# B&R Automation Studio project 02_BASE_PROJECT
Automation Studio 4.9

## Configuration Config1

CPU X20CP1382, AutomationRuntime A4.83, Build 4.1.2, Safety 0.0, Vc V4.73.2

### Task classes (Cpu.sw)
```
Cyclic#1 (cycle 2000 us, tolerance 0 us):
  ComTCP_P <- Libraries.ComTCP.ComTCP_P.prg
  Input_Brid <- Input_Bridge.prg
  Output_Bri <- Output_Bridge.prg
  PLCopen <- PLCopen.prg [disabled]
Cyclic#2:
  LED_IO <- LED_IO.prg
  Master <- Master.prg
  Slave <- Slave.prg
DataObjects: Acp10sys
NcDataObjects: acp10etxen <- acp10etxen.dob, gAxis01a <- gAxis01obj.gAxis01a.dob, gAxis01i <- gAxis01obj.gAxis01i.dob, gAxis02a <- gAxis02obj.gAxis02a.dob, gAxis02i <- gAxis02obj.gAxis02i.dob, MyCam <- MyCam.dob, MyCamBis <- MyCamBis.dob
Binaries: udbdef, FWRules, TCData, arsvcreg, mvLoader, TCLang, acp10cfg, Acp10map, sysconf, Role, User, iomap, ashwd, asfw, arconfig, ashwac, Config, TC
Libraries: Acp10man, Acp10par, NcGlobal, Acp10_MC, sys_lib, brsystem, runtime, Acp10sim, MpAxis, MpBase, MpCom, AsTCP, standard, AsArLog, AsBrStr, ComTCP_L, operator, astime, AsIecCon, My_Library, AsIODiag, fileio, powerlnk, dataobj, arssl
```

### Hardware
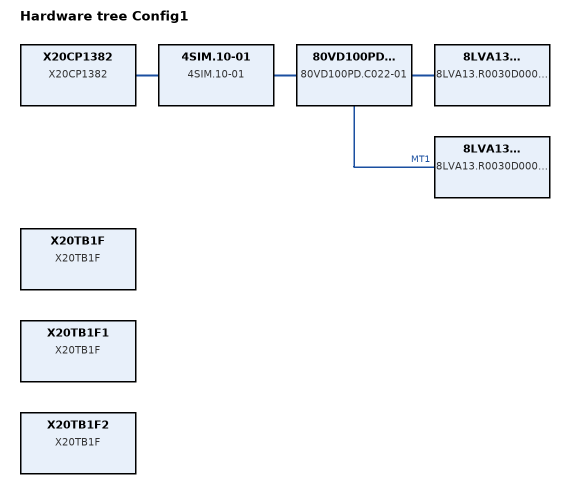
```
4SIM.10-01 : 4SIM.10-01 v1.3.0.0  [PLK1 -> X20CP1382.IF3 (NodeNumber=1) [Cable Type=PowerlinkCable, Length=10, Version=1.0.0.3]; PLK2 -> 80VD100PD.C022-01.PLK1 (NodeNumber=1) [Cable Type=PowerlinkCable, Length=10, Version=1.0.0.3]]
  Supervision = off
80VD100PD.C022-01 : 80VD100PD.C022-01 v2.5.0.0  [PLK1 -> 4SIM.10-01.PLK2 (NodeNumber=2) [Cable Type=PowerlinkCable, Length=10, Version=1.0.0.3]; MT2 -> 8LVA13.R0030D000-0.MT]
  MotionTP = Acp10Arnc0
  AxisIsPeriodic_r1 = on
  Period_r1 = 360
  BothEndSwitchesAreNormallyOpen_r1 = on
  QuickStopIsNormallyOpen_r1 = on
  AxisIsPeriodic_r2 = on
  Period_r2 = 360
  BothEndSwitchesAreNormallyOpen_r2 = on
  QuickStopIsNormallyOpen_r2 = on
8LVA13.R0030D000-0 : 8LVA13.R0030D000-0 v2.2.0.4  [MT -> 80VD100PD.C022-01.MT2]
8LVA13.R0030D000-0a : 8LVA13.R0030D000-0 v2.2.0.4  [MT -> 80VD100PD.C022-01.MT1]
X20CP1382 : X20CP1382 v1.14.0.0  [X1 -> X1.SL; X2 -> X2.SL; X3 -> X3.SL]
  Module X1 (Type=X1, Virtual=true, Version=1.14.0.0)
    Connection (Connector=SS1, TargetModule=X20TB1F, TargetConnector=SS)
    Connection (Connector=SL, TargetModule=X20CP1382, TargetConnector=X1)
  Module X2 (Type=X2, Virtual=true, Version=1.14.0.0)
    Connection (Connector=SS1, TargetModule=X20TB1F1, TargetConnector=SS)
    Connection (Connector=SL, TargetModule=X20CP1382, TargetConnector=X2)
  Module X3 (Type=X3, Virtual=true, Version=1.14.0.0)
    Connection (Connector=SS1, TargetModule=X20TB1F2, TargetConnector=SS)
    Connection (Connector=SL, TargetModule=X20CP1382, TargetConnector=X3)
  Connector IF2:
    ActivateDevice = 1
    Mode = Manual
    InternetAddress = 192.168.0.1
    SubnetMask = 255.255.255.0
    ActivateSnmp = 2
  Connector IF3:
    CycleTime = 2000
  ConfigurationID = UniboTest2024_Config1
  Simulation = 1
  TimerDeviceType = EPLX2X
  TimerDevice = X20CP1382.IF3
  TaskClassIdleTime = 6000
  Cyclic1Duration = 2000
  Cyclic1Tolerance = 0
  ActivateOpcUa = 1
  OpcUaInformationModels_PV_Version = 1
X20TB1F : X20TB1F v1.0.0.0
X20TB1F1 : X20TB1F v1.0.0.0
X20TB1F2 : X20TB1F v1.0.0.0
```

### Acp10map.ncm - X20CP1382/Motion/Acp10map.ncm
```
NcMapping (NcSwId=Acp10)
  NcObject gAxis01 (ModuleId=80VD100PD.C022-01, Type=ncAXIS, Channel=1, AcoposSimulation=Off, InitParameter=gAxis01i, AcoposParameter=gAxis01a, AdditionalData=PLCopen_ModPos="360,1" , Disabled=FALSE, ModuleDisabled=FALSE)
  NcObject gAxis02 (ModuleId=80VD100PD.C022-01, Type=ncAXIS, Channel=2, AcoposSimulation=Off, InitParameter=gAxis02i, AcoposParameter=gAxis02a, AdditionalData=PLCopen_ModPos="360,1" , Disabled=FALSE, ModuleDisabled=FALSE)
  NcObject 80VD100PD.C022-01_ncV_AXIS1 (ModuleId=80VD100PD.C022-01, Type=ncV_AXIS, Channel=1, Disabled=TRUE, ModuleDisabled=FALSE)
  NcObject 80VD100PD.C022-01_ncV_AXIS2 (ModuleId=80VD100PD.C022-01, Type=ncV_AXIS, Channel=2, Disabled=TRUE, ModuleDisabled=FALSE)
```

## Logical view

Binary libraries used (declarations not repeated): operator, runtime, astime, AsIecCon, sys_lib, brsystem, MpAxis, AsTCP, standard, AsArLog, AsBrStr, MpBase, MpCom, AsIODiag, Acp10man, Acp10par, NcGlobal, Acp10sim 5.24.1, Acp10_MC

### Global.var
```iecst
(*Name of Axis*)
VAR
	gAxis01 : ACP10AXIS_typ;
	gAxis02 : ACP10AXIS_typ;
END_VAR
(*Hardware Variables*)
VAR
	Conv_Lock : BOOL;
	Cutter_Lock : BOOL;
	Start_Button : BOOL;
	Stop_Button : BOOL;
	Sensor_Button : BOOL;
	Reset_Button : BOOL;
	Speed : INT;
	Position : INT;
	DI1 : FSM_LED;
	DI2 : FSM_LED;
	DI3 : FSM_LED;
	DI4 : FSM_LED;
	DI5 : FSM_LED;
	DI6 : FSM_LED;
	Display : INT;
END_VAR
(*HMI Variables*)
VAR
	Emergancy_Button_HMI : BOOL;
	Start_Button_HMI : BOOL;
	Stop_Button_HMI : BOOL;
	Sensor_Button_HMI : BOOL;
	Reset_Button_HMI : BOOL;
	Conv_Lock_HMI : BOOL;
	Cutter_Lock_HMI : BOOL;
	Conv_Speed_HMI : REAL;
	Cutter_Speed_HMI : REAL;
	Cutting_Pos_HMI : REAL;
	Cutting_Depth_HMI : REAL;
	Blade_Up_Man_HMI : BOOL;
	Blade_Down_Man_HMI : BOOL;
	Conv_Right_Man_HMI : BOOL;
	Conv_Left_Man_HMI : BOOL;
	Slow_Blade_HMI : BOOL;
	Slow_Conv_HMI : BOOL;
	LED_DI1_HMI : BOOL;
	LED_DI2_HMI : BOOL;
	LED_DI3_HMI : BOOL;
	LED_DI4_HMI : BOOL;
	LED_DI5_HMI : BOOL;
	LED_DI6_HMI : BOOL;
	Dis_Conv_Speed_HMI : REAL;
	Dis_Cut_Speed_HMI : REAL;
	Dis_Cut_Pos_HMI : INT;
	Dis_Cut_Depth_HMI : INT;
	Man_Mode_HMI : BOOL;
	Over_Ride_HMI : BOOL;
END_VAR
(*LED_IO Variables*)
VAR
	Power_Axis : BOOL;
	Home_Axis : BOOL;
	Reset_Command : BOOL;
	Error_Command : BOOL;
	Start_Command : BOOL := FALSE;
	Stop_Command : BOOL := FALSE;
END_VAR
(*Master Variables*)
VAR
	Do_Cut : BOOL;
	Done_Cut : BOOL;
	Master : MpAxisBasic;
	M_Active : BOOL;
	M_Error : BOOL;
	M_Actual_Position : LREAL;
	M_Actual_Velocity : LREAL;
	M_Homed : BOOL;
	M_Powered : BOOL;
	M_Stoped : BOOL;
END_VAR
(*Slave Variables*)
VAR
	Slave : MpAxisBasic;
	Coupling : MpAxisCoupling;
	S_Active : BOOL;
	S_Error : BOOL;
	S_Homed : BOOL;
	S_Powered : BOOL;
	C_Error : BOOL;
	S_Actual_Position : LREAL;
	S_Actual_Velocity : LREAL;
	S_Stoped : BOOL;
END_VAR
(*Input Bridige Variables*)
VAR
	Conv_Speed : REAL;
	Start_Trigger : BOOL;
	Stop_Trigger : BOOL;
	Error_Trigger : BOOL;
	Reset_Trigger : BOOL;
	Conv_Lock_HMI_Trigger : BOOL;
	Cutter_Lock_HMI_Trigger : BOOL;
	Sensor_Trigger : BOOL;
	Conv_Lock_Trigger : BOOL;
	Over_Ride_Trigger : BOOL;
	Cutter_Lock_Trigger : BOOL;
	Slow_Blade_Trigger : BOOL;
	Blade_Up_Man_HMI_Trigger : BOOL;
	Blade_Down_Man_HMI_Trigger : BOOL;
	Conv_Left_Man_HMI_Trigger : BOOL;
	Conv_Right_Man_HMI_Trigger : BOOL;
	Slow_Conv_Trigger : BOOL;
END_VAR
(*Manual Motion Variables*)
VAR
	Manual_Mode_Trigger : BOOL;
	Man_Mode_OFF : BOOL := TRUE;
	Blade_Jog_Velocity : REAL;
	Conv_Jog_Velocity : REAL;
END_VAR
```

- Project.language (not shown)

### Data object Logical/acp10etxen (Ett)

- acp10etxen.ett (not shown)

### Data object Logical/gAxis01obj/gAxis01a (Apt)

#### gAxis01a.apt
```
AcoposParameterTable:
  Root Parameters
```

### gAxis01i.ax
```
InitParameter (Version=5.20.1, NcSwId=ACP10)
  ACP10AXIS_typ:
    dig_in:
      level:
        reference = ncACTIV_HI
        pos_hw_end = ncACTIV_HI
        neg_hw_end = ncACTIV_HI
        trigger1 = ncACTIV_HI
        trigger2 = ncACTIV_HI
    encoder_if:
      parameter:
        count_dir = ncSTANDARD
        scaling:
          load:
            units = 360
            rev_motor = 1
    limit:
      parameter:
        v_pos = 10000.0
        v_neg = 10000.0
        a1_pos = 50000.0
        a2_pos = 50000.0
        a1_neg = 50000.0
        a2_neg = 50000.0
        t_jolt = 0.0
        t_in_pos = 0.0
        pos_sw_end = 2000000000
        neg_sw_end = -2000000000
        ds_warning = 500.0
        ds_stop = 1000.0
        a_stop = 1.0E+30
        dv_stop = 0.0
        dv_stop_mode = ncOFF
    controller:
      mode = ncPOSITION
      position:
        kv = 289.0
        tn = 0.0
        t_predict = 0.0004
        t_total = 0.0004
        p_max = 1.0E+30
        i_max = 0.0
      speed:
        kv = 0.9
        tn = 0.0
        t_filter = 0.0
        isq_filter1:
          type = ncOFF
          a0 = 0.0
          a1 = 0.0
          b0 = 0.0
          b1 = 0.0
          b2 = 0.0
          c0_par_id = 0
          c1_par_id = 0
        isq_filter2:
          type = ncOFF
          a0 = 0.0
          a1 = 0.0
          b0 = 0.0
          b1 = 0.0
          b2 = 0.0
          c0_par_id = 0
          c1_par_id = 0
        isq_filter3:
          type = ncOFF
          a0 = 0.0
          a1 = 0.0
          b0 = 0.0
          b1 = 0.0
          b2 = 0.0
          c0_par_id = 0
          c1_par_id = 0
      uf:
        type = ncLINEAR + ncCORRECTION
        auto_config = ncMOTOR_PAR
        u0 = 0.0
        un = 0.0
        fn = 50.0
        k_f_slip = 0.0
      ff:
        mode = ncSTANDARD
        torque_load = 0.0
        torque_pos = 0.0
        torque_neg = 0.0
        kv_torque = 0.0
        inertia = 0.0
        t_filter_a = 0.0
      fb:
        mode = ncSTANDARD
        speed_mix_ratio = 0.0
        speed_kv = 0.0
      model:
        mass1:
          inertia = 0.0
          viscous_friction = 0.0
        mass2:
          inertia = 0.0
          viscous_friction = 0.0
          stiffness = 0.0
          damping = 0.0
    move:
      stop:
        parameter[0]:
          decel_ramp = ncA_LIMIT
          controller = ncON
        parameter[1]:
          decel_ramp = ncA_LIMIT
          controller = ncON
        parameter[2]:
          decel_ramp = ncA_LIMIT
          controller = ncON
        parameter[3]:
          decel_ramp = ncA_LIMIT
          controller = ncON
        quickstop:
          decel_ramp = ncA_LIMIT
          t_jolt = 0.0
        drive_error:
          decel_ramp = ncA_LIMIT
      homing:
        parameter:
          s = 0
          v_switch = 5000.0
          v_trigger = 500.0
          a = 50000.0
          mode = ncDIRECT
          edge_sw = ncPOSITIVE
          start_dir = ncPOSITIVE
          trigg_dir = ncPOSITIVE
          ref_pulse = ncOFF
          fix_dir = ncOFF
          tr_s_block = 0.0
          torque_lim = 0.0
          ds_block = 0.0
          ds_stop = 0.0
      basis:
        parameter:
          v_pos = 5000.0
          v_neg = 5000.0
          a1_pos = 50000.0
          a2_pos = 50000.0
          a1_neg = 50000.0
          a2_neg = 50000.0
    message:
      text:
        parameter:
          format = ncBREAK
          columns = 80
          data_modul = acp10etxen
```

- Data object Logical/gAxis02obj/gAxis02a (Apt) (no source held here)

### gAxis02i.ax
```
InitParameter (Version=5.20.1, NcSwId=Acp10)
  ACP10AXIS_typ:
    dig_in:
      level:
        reference = ncACTIV_HI
        pos_hw_end = ncACTIV_HI
        neg_hw_end = ncACTIV_HI
        trigger1 = ncACTIV_HI
        trigger2 = ncACTIV_HI
    encoder_if:
      parameter:
        count_dir = ncSTANDARD
        scaling:
          load:
            units = 360
            rev_motor = 1
    limit:
      parameter:
        v_pos = 10000
        v_neg = 10000
        a1_pos = 50000
        a2_pos = 50000
        a1_neg = 50000
        a2_neg = 50000
        t_jolt = 0
        t_in_pos = 0
        pos_sw_end = 2000000000
        neg_sw_end = -2000000000
        ds_warning = 500
        ds_stop = 1000
        a_stop = 1.0e30
        dv_stop = 0
        dv_stop_mode = ncOFF
    controller:
      mode = ncPOSITION
      position:
        kv = 289.0
        tn = 0
        t_predict = 0.0004
        t_total = 0.0004
        p_max = 1.0e30
        i_max = 0
      speed:
        kv = 0.9
        tn = 0
        t_filter = 0.0
        isq_filter1:
          type = ncOFF
          a0 = 0.0
          a1 = 0.0
          b0 = 0.0
          b1 = 0.0
          b2 = 0.0
          c0_par_id = 0
          c1_par_id = 0
        isq_filter2:
          type = ncOFF
          a0 = 0.0
          a1 = 0.0
          b0 = 0.0
          b1 = 0.0
          b2 = 0.0
          c0_par_id = 0
          c1_par_id = 0
        isq_filter3:
          type = ncOFF
          a0 = 0.0
          a1 = 0.0
          b0 = 0.0
          b1 = 0.0
          b2 = 0.0
          c0_par_id = 0
          c1_par_id = 0
      uf:
        type = ncLINEAR + ncCORRECTION
        auto_config = ncMOTOR_PAR
        u0 = 0
        un = 0
        fn = 50.0
        k_f_slip = 0
      ff:
        mode = ncSTANDARD
        torque_load = 0.0
        torque_pos = 0.0
        torque_neg = 0.0
        kv_torque = 0.0
        inertia = 0.0
        t_filter_a = 0.0
      fb:
        mode = ncSTANDARD
        speed_mix_ratio = 0.0
        speed_kv = 2.0
      model:
        mass1:
          inertia = 0
          viscous_friction = 0
        mass2:
          inertia = 0
          viscous_friction = 0
          stiffness = 0
          damping = 0
    move:
      stop:
        parameter[0]:
          decel_ramp = ncA_LIMIT
          controller = ncON
        parameter[1]:
          decel_ramp = ncA_LIMIT
          controller = ncON
        parameter[2]:
          decel_ramp = ncA_LIMIT
          controller = ncON
        parameter[3]:
          decel_ramp = ncA_LIMIT
          controller = ncON
        quickstop:
          decel_ramp = ncA_LIMIT
          t_jolt = 0
        drive_error:
          decel_ramp = ncA_LIMIT
      homing:
        parameter:
          s = 0
          v_switch = 5000
          v_trigger = 500
          a = 50000
          mode = ncDIRECT
          edge_sw = ncPOSITIVE
          start_dir = ncPOSITIVE
          trigg_dir = ncPOSITIVE
          ref_pulse = ncOFF
          fix_dir = ncOFF
          tr_s_block = 0
          torque_lim = 0
          ds_block = 0
          ds_stop = 0
      basis:
        parameter:
          v_pos = 5000
          v_neg = 5000
          a1_pos = 50000
          a2_pos = 50000
          a1_neg = 50000
          a2_neg = 50000
    message:
      text:
        parameter:
          format = ncBREAK
          columns = 80
          data_modul = acp10etxen
```

### Program Logical/Input_Bridge

#### Main.st
```iecst
PROGRAM _INIT
	(* Insert code here *)
	//Initial Parameters

	Conv_Speed 		:= 100.0;

END_PROGRAM

PROGRAM _CYCLIC

	IF DiagCpuIsSimulated() THEN
		(* For Simulation *)
		//Operator
		//LED_IO Bridge
		Start_Trigger 			:= ComTCP_SimInputs.Start_Button_ButtonPress 		OR Start_Button_HMI;
		Stop_Trigger 			:= ComTCP_SimInputs.Stop_Button_ButtonPress 		OR Stop_Button_HMI;
		Error_Trigger 			:= ComTCP_SimInputs.Emergency_Button_ButtonToggle 	OR Emergancy_Button_HMI OR M_Error OR S_Error OR C_Error;
		Reset_Trigger 			:= ComTCP_SimInputs.White_Button_ButtonPress 		OR Reset_Button_HMI;
		Sensor_Trigger 			:= ComTCP_SimInputs.Yellow_Button_ButtonPress 		OR Sensor_Button_HMI;
		Conv_Lock_HMI_Trigger 	:= Conv_Lock_HMI;
		Cutter_Lock_HMI_Trigger := Cutter_Lock_HMI;

		IF Conv_Lock_HMI_Trigger THEN
			IF Conv_Speed_HMI < 10 THEN
				Conv_Speed 	:= 10;
			ELSE
				Conv_Speed 	:= Conv_Speed_HMI;
			END_IF
		END_IF

		//Manual Motion
		Manual_Mode_Trigger 		:= Man_Mode_HMI;
		Slow_Blade_Trigger 			:= Slow_Blade_HMI;
		Slow_Conv_Trigger 			:= Slow_Conv_HMI;
		Blade_Up_Man_HMI_Trigger 	:= Blade_Up_Man_HMI;
		Blade_Down_Man_HMI_Trigger 	:= Blade_Down_Man_HMI;
		Conv_Left_Man_HMI_Trigger 	:= Conv_Left_Man_HMI;
		Conv_Right_Man_HMI_Trigger 	:= Conv_Right_Man_HMI;

		IF Slow_Blade_Trigger THEN
			Blade_Jog_Velocity := 5.0;
		ELSE
			Blade_Jog_Velocity := 100.0;
		END_IF

		IF Slow_Conv_Trigger THEN
			Conv_Jog_Velocity := 5.0;
		ELSE
			Conv_Jog_Velocity := 100.0;
		END_IF

	ELSE
		(* For Actual Setup *)
		Start_Trigger 			:= Start_Button 		OR Start_Button_HMI;
		Stop_Trigger 			:= Stop_Button 			OR Stop_Button_HMI;
		Error_Trigger 			:= Emergancy_Button_HMI OR M_Error OR S_Error;
		Reset_Trigger 			:= Reset_Button 		OR Reset_Button_HMI;
		Sensor_Trigger 			:= Sensor_Button 		OR Sensor_Button_HMI;
		Conv_Lock_HMI_Trigger	:= Conv_Lock_HMI;
		Conv_Lock_HMI_Trigger 	:= Conv_Lock;
		Over_Ride_Trigger 		:= Over_Ride_HMI;
		IF Over_Ride_Trigger THEN
			IF Conv_Lock_HMI_Trigger THEN
				IF Conv_Speed_HMI < 10 THEN
					Conv_Speed 	:= 10;
				ELSE
					Conv_Speed 	:= Conv_Speed_HMI;
				END_IF
			END_IF
		ELSE
			IF Conv_Lock_Trigger THEN
				Conv_Speed 		:= (Speed*3000/32767);
			END_IF
		END_IF

		//Manual Motion
		Manual_Mode_Trigger 		:= Man_Mode_HMI;
		Slow_Blade_Trigger 			:= Slow_Blade_HMI;
		Slow_Conv_Trigger 			:= Slow_Conv_HMI;
		Blade_Up_Man_HMI_Trigger 	:= Blade_Up_Man_HMI;
		Blade_Down_Man_HMI_Trigger 	:= Blade_Down_Man_HMI;
		Conv_Left_Man_HMI_Trigger	:= Conv_Left_Man_HMI;
		Conv_Right_Man_HMI_Trigger 	:= Conv_Right_Man_HMI;
		IF Slow_Blade_Trigger THEN
			Blade_Jog_Velocity := 5.0;
		ELSE
			Blade_Jog_Velocity := 100.0;
		END_IF

		IF Slow_Conv_Trigger THEN
			Conv_Jog_Velocity := 5.0;
		ELSE
			Conv_Jog_Velocity := 100.0;
		END_IF

	END_IF

END_PROGRAM

PROGRAM _EXIT
	(* Insert code here *)

END_PROGRAM
```

### Program Logical/LED_IO

#### Main.st
```iecst
PROGRAM _INIT
	(* Insert code here *)

END_PROGRAM

PROGRAM _CYCLIC
	(* Insert code here *)
	CASE State OF
		0: //Initiation
			DI1(LED_State := 'off');
			DI2(LED_State := 'off');
			DI3(LED_State := 'off');
			DI4(LED_State := 'off');
			DI5(LED_State := 'off');
			DI6(LED_State := 'off');

			IF M_Active AND S_Active AND Man_Mode_OFF THEN
				State := 2;
			END_IF

		1: //Error

			DI1(LED_State := 'off');
			DI2(LED_State := 'off');
			DI3(LED_State := 'off');
			DI4(LED_State := 'off');
			DI5(LED_State := 'off');
			DI6(LED_State := 'blink');

			Error_Command 	:= TRUE;
			Start_Command 	:= FALSE;
			Stop_Command 	:= TRUE;
			Power_Axis 		:= FALSE;

			IF Reset_Trigger THEN
				Reset_Command 	:= TRUE;
				IF NOT Error_Trigger THEN
					Reset_Command 	:= FALSE;
					State 			:= 2;
				END_IF
			END_IF

		2: //Disabled

			DI1(LED_State := 'on');
			DI2(LED_State := 'on');
			DI3(LED_State := 'on');
			DI4(LED_State := 'on');
			DI5(LED_State := 'on');
			DI6(LED_State := 'on');

			IF Reset_Trigger THEN
				Power_Axis 	:= TRUE;
			END_IF

			IF Error_Trigger THEN
				State := 1;
			END_IF

			IF M_Powered AND S_Powered AND NOT (M_Homed AND S_Homed) THEN
				State := 3;
			END_IF

			IF M_Powered AND S_Powered AND M_Homed AND S_Homed THEN
				State := 4;
			END_IF

			IF NOT Man_Mode_OFF THEN
				State := 0;
			END_IF

		3: //Homing
			DI1(LED_State := 'blink');
			DI2(LED_State := 'blink');
			DI3(LED_State := 'blink');
			DI4(LED_State := 'blink');
			DI5(LED_State := 'blink');
			DI6(LED_State := 'blink');

			Home_Axis := TRUE;

			IF M_Homed AND S_Homed THEN
				Home_Axis 	:= FALSE;
				State 		:= 4;
			END_IF

			IF Error_Trigger THEN
				State := 1;
			END_IF

			IF NOT Man_Mode_OFF THEN
				State := 0;
			END_IF

		4://Ready
			IF NOT (Conv_Lock_Trigger OR Conv_Lock_HMI_Trigger) THEN
				DI1(LED_State := 'off');
			END_IF
			IF NOT (Cutter_Lock_Trigger OR Cutter_Lock_HMI_Trigger) THEN
				DI2(LED_State := 'off');
			END_IF
			IF (Conv_Lock_Trigger OR Conv_Lock_HMI_Trigger) THEN
				DI1(LED_State := 'on');
			END_IF
			IF (Cutter_Lock_Trigger OR Cutter_Lock_HMI_Trigger) THEN
				DI2(LED_State := 'on');
			END_IF

			DI3(LED_State := 'blink');
			DI4(LED_State := 'off');
			DI5(LED_State := 'off');
			DI6(LED_State := 'off');

			Error_Command 	:= FALSE;
			Power_Axis 		:= TRUE;

			IF Start_Trigger AND NOT Error_Trigger THEN
				State := 5;
			END_IF

			IF Error_Trigger THEN
				State := 1;
			END_IF

			IF NOT Man_Mode_OFF THEN
				State := 0;
			END_IF

		5://Run
			IF NOT (Conv_Lock_Trigger OR Conv_Lock_HMI_Trigger) THEN
				DI1(LED_State := 'off');
			END_IF
			IF NOT (Cutter_Lock_Trigger OR Cutter_Lock_HMI_Trigger) THEN
				DI2(LED_State := 'off');
			END_IF
			IF (Conv_Lock_Trigger OR Conv_Lock_HMI_Trigger) THEN
				DI1(LED_State := 'on');
			END_IF
			IF (Cutter_Lock_Trigger OR Cutter_Lock_HMI_Trigger) THEN
				DI2(LED_State := 'on');
			END_IF

			DI3(LED_State := 'on');
			DI4(LED_State := 'on');
			DI5(LED_State := 'off');
			DI6(LED_State := 'off');

			Start_Command 	:= TRUE;
			Stop_Command 	:= FALSE;
			Power_Axis 		:= TRUE;

			IF Error_Trigger THEN
				State := 1;
			END_IF

			IF Stop_Trigger AND NOT Error_Trigger THEN
				State := 6;
			END_IF

			IF NOT Man_Mode_OFF THEN
				State := 0;
			END_IF

		6://Stop

			Start_Command 	:= FALSE;
			Stop_Command 	:= TRUE;

			IF M_Stoped THEN
				Stop_Command 	:= FALSE;
				State 			:= 4;
			END_IF

			IF Error_Trigger THEN
				State := 1;
			END_IF

			IF NOT Man_Mode_OFF THEN
				State := 0;
			END_IF

	END_CASE

END_PROGRAM

PROGRAM _EXIT
	(* Insert code here *)

END_PROGRAM
```

### Program Logical/Libraries/ComTCP/ComTCP_L

#### MNG_Global.hpp
```cpp
#ifndef  _MNGGLOBAL_HPP_
#define _MNGGLOBAL_HPP_

#include <mng_globalTYP.h>

    typedef struct {

		signed short NumSignals;

        /* BOOL Emergency_Button_ButtonToggle */
        BOOL Emergency_Button_ButtonToggle;
        /* BOOL Yellow_Button_ButtonPress */
        BOOL Yellow_Button_ButtonPress;
        /* BOOL White_Button_ButtonPress */
        BOOL White_Button_ButtonPress;
        /* BOOL Start_Button_ButtonPress */
        BOOL Start_Button_ButtonPress;
        /* BOOL Stop_Button_ButtonPress */
        BOOL Stop_Button_ButtonPress;
        /* REAL Knob_0_AXIS */
        REAL Knob_0_AXIS;
        /* REAL Knob_1_AXIS */
        REAL Knob_1_AXIS;
        /* REAL Knob_2_AXIS */
        REAL Knob_2_AXIS;
        /* REAL Knob_3_AXIS */
        REAL Knob_3_AXIS;
        /* REAL Shaft_1_AXIS */
        REAL Shaft_1_AXIS;
        /* BOOL Shaft_1_LBK */
        BOOL Shaft_1_LBK;
        /* BOOL Shaft_1_LFR */
        BOOL Shaft_1_LFR;
        /* REAL Shaft_0_AXIS */
        REAL Shaft_0_AXIS;
        /* BOOL Shaft_0_LBK */
        BOOL Shaft_0_LBK;
        /* BOOL Shaft_0_LFR */
        BOOL Shaft_0_LFR;

        } ComTCP_INPUTS_32BIT_FWRD;

    typedef struct {

		signed short NumSignals;

        /* UDINT Yellow_light_Key */
        UDINT Yellow_light_Key;
        /* UDINT Stop_light_Key */
        UDINT Stop_light_Key;
        /* UDINT White_light_Key */
        UDINT White_light_Key;
        /* UDINT Green_light_Key */
        UDINT Green_light_Key;
        /* REAL Shaft_0_ACT_POS */
        REAL Shaft_0_ACT_POS;
        /* REAL Shaft_1_ACT_POS */
        REAL Shaft_1_ACT_POS;

        } ComTCP_OUTPUTS_32BIT_FWRD;

#endif
```

#### MNG_CpyMsgToInp.cpp
```cpp
#include "MNG_InternalTyp.hpp"

unsigned long int MNG_CpyMsgToInp(MNG_RawDatagram * pFromServer, ComTCP_INPUTS_32BIT_FWRD *pSimInputs) {

    MNG_DatagramType datagramType;
	unsigned long int DWordBuffer;
        unsigned long int byteCount;
	unsigned long int numSignalsInMessage;

	byteCount = N_TO_HUDINT((pFromServer->Header).ByteCount);
	datagramType = static_cast<MNG_DatagramType>(N_TO_HUDINT((pFromServer->Header).DatagramType));
	if (datagramType != MNG_Raw32BitImage) {
		return 0;
	}

    pSimInputs->NumSignals = 15;

    numSignalsInMessage = N_TO_HUDINT(pFromServer->Payload[0]);
        if ((static_cast<long int>(numSignalsInMessage) != pSimInputs->NumSignals) ||
	(byteCount != 4 + numSignalsInMessage * 4)) {
		return 0;
	}

    /* BOOL Emergency_Button_ButtonToggle */
    pSimInputs->Emergency_Button_ButtonToggle = (pFromServer->Payload[1] != 0);

    /* BOOL Yellow_Button_ButtonPress */
    pSimInputs->Yellow_Button_ButtonPress = (pFromServer->Payload[2] != 0);

    /* BOOL White_Button_ButtonPress */
    pSimInputs->White_Button_ButtonPress = (pFromServer->Payload[3] != 0);

    /* BOOL Start_Button_ButtonPress */
    pSimInputs->Start_Button_ButtonPress = (pFromServer->Payload[4] != 0);

    /* BOOL Stop_Button_ButtonPress */
    pSimInputs->Stop_Button_ButtonPress = (pFromServer->Payload[5] != 0);

    /* FLOAT32 Knob_0_AXIS */
    DWordBuffer = N_TO_HUDINT(pFromServer->Payload[6]);
    brsmemcpy((unsigned long int)&(pSimInputs->Knob_0_AXIS), (unsigned long int)&(DWordBuffer), 4);

    /* FLOAT32 Knob_1_AXIS */
    DWordBuffer = N_TO_HUDINT(pFromServer->Payload[7]);
    brsmemcpy((unsigned long int)&(pSimInputs->Knob_1_AXIS), (unsigned long int)&(DWordBuffer), 4);

    /* FLOAT32 Knob_2_AXIS */
    DWordBuffer = N_TO_HUDINT(pFromServer->Payload[8]);
    brsmemcpy((unsigned long int)&(pSimInputs->Knob_2_AXIS), (unsigned long int)&(DWordBuffer), 4);

    /* FLOAT32 Knob_3_AXIS */
    DWordBuffer = N_TO_HUDINT(pFromServer->Payload[9]);
    brsmemcpy((unsigned long int)&(pSimInputs->Knob_3_AXIS), (unsigned long int)&(DWordBuffer), 4);

    /* FLOAT32 Shaft_1_AXIS */
    DWordBuffer = N_TO_HUDINT(pFromServer->Payload[10]);
    brsmemcpy((unsigned long int)&(pSimInputs->Shaft_1_AXIS), (unsigned long int)&(DWordBuffer), 4);

    /* BOOL Shaft_1_LBK */
    pSimInputs->Shaft_1_LBK = (pFromServer->Payload[11] != 0);

    /* BOOL Shaft_1_LFR */
    pSimInputs->Shaft_1_LFR = (pFromServer->Payload[12] != 0);

    /* FLOAT32 Shaft_0_AXIS */
    DWordBuffer = N_TO_HUDINT(pFromServer->Payload[13]);
    brsmemcpy((unsigned long int)&(pSimInputs->Shaft_0_AXIS), (unsigned long int)&(DWordBuffer), 4);

    /* BOOL Shaft_0_LBK */
    pSimInputs->Shaft_0_LBK = (pFromServer->Payload[14] != 0);

    /* BOOL Shaft_0_LFR */
    pSimInputs->Shaft_0_LFR = (pFromServer->Payload[15] != 0);

return N_TO_HUDINT((pFromServer->Header).Counter); // return counter
}
```

### Library Logical/Libraries/My_Library (IEC)

#### My_Library.fun - Exported functions and function blocks
```iecst
FUNCTION_BLOCK FSM_LED
	VAR_INPUT
		LED_State : STRING[80];
	END_VAR
	VAR_OUTPUT
		LED_Light : BOOL;
	END_VAR
	VAR
		Timer : TON;
		State : INT := 0;
	END_VAR
END_FUNCTION_BLOCK

FUNCTION_BLOCK FSM_AXIS (*For Motion of the motors*)
	VAR_INPUT
		Axis_Name : UDINT;
		Deceleration : REAL;
		Velocity : REAL;
		Acceleration : REAL;
		Direction : USINT;
		Distance : REAL;
		Position : REAL;
		Home : BOOL;
		Power : BOOL;
		Move_Velocity : BOOL;
		Move_Absolute : BOOL;
		Move_Additive : BOOL;
		Stop : BOOL;
		Reset_Error : BOOL;
	END_VAR
	VAR_OUTPUT
		Actual_Position : REAL;
		Actual_Velocity : REAL;
		Active : BOOL;
		Power_ON : BOOL;
		Stop_Done : BOOL;
		Is_Homed : BOOL;
		Move_Abs_Done : BOOL;
		Move_Add_Done : BOOL;
		Error : BOOL; (*Code Parameters*)
	END_VAR
	VAR
		MCRS : MC_ReadStatus; (*List of all the PLCOpen libraries*)
		RS_Valid : BOOL;
		RS_Error : BOOL;
		RS_Errorstop : BOOL;
		RS_Disabled : BOOL;
		MCP : MC_Power;
		P_Enable : BOOL;
		P_Status : BOOL;
		P_Error : BOOL;
		MCH : MC_Home;
		H_Execute : BOOL;
		H_Done : BOOL;
		H_Error : BOOL;
		MCS : MC_Stop;
		S_Execute : BOOL;
		S_Done : BOOL;
		S_Error : BOOL;
		MCR : MC_Reset;
		R_Execute : BOOL;
		R_Done : BOOL;
		R_Error : BOOL;
		MCRAP : MC_ReadActualPosition;
		RAP_Valid : BOOL;
		RAP_Error : BOOL;
		MCRAV : MC_ReadActualVelocity;
		RAV_Valid : BOOL;
		RAV_Error : BOOL;
		MCMV : MC_MoveVelocity;
		V_Execute : BOOL;
		V_Error : BOOL;
		MCMAdd : MC_MoveAdditive;
		Add_Execute : BOOL;
		Add_Done : BOOL;
		Add_Error : BOOL;
		MCMA : MC_MoveAbsolute;
		A_Execute : BOOL;
		A_Done : BOOL;
		A_Error : BOOL;
		State : INT := 0;
		Move_Absolute_Old : BOOL;
		Move_Additive_Old : BOOL;
		Old_Velocity : REAL;
	END_VAR
END_FUNCTION_BLOCK
```

### Program Logical/Master

#### Variables.var
```iecst
VAR
	Master_Param : MpAxisBasicParType;
	State : USINT := 0;
	M_Update : BOOL;
	M_MoveVelocity : BOOL;
	M_MoveAbsolute : BOOL;
	M_MoveAdditive : BOOL;
	M_Velocity : REAL;
	M_Stop : BOOL;
	M_Jog_Param : MpAxisJogType;
	M_Jog_Positive : BOOL;
	M_Jog_Negative : BOOL;
END_VAR
```

#### Main.st
```iecst
PROGRAM _INIT
	(* Insert code here *)
	Master_Param.Acceleration := 10000;
	Master_Param.Deceleration := 10000;

END_PROGRAM

PROGRAM _CYCLIC

	IF Sensor_Trigger THEN
		Do_Cut 	:= TRUE;
	END_IF

	IF Do_Cut AND Done_Cut THEN
		Do_Cut 		:= FALSE;
		Done_Cut 	:= FALSE;
	END_IF

	CASE State OF
		0: //Standstill
			M_MoveVelocity := FALSE;
			M_Stop:= FALSE;
			IF NOT Error_Command AND Start_Command AND Man_Mode_OFF THEN
				State := 1;
			END_IF

			IF Manual_Mode_Trigger THEN
				State := 2;
			END_IF

		1://Moving Conveyor
			M_MoveVelocity 	:= TRUE;
			M_Stop			:= FALSE;
			M_Jog_Positive 	:= FALSE;
			M_Jog_Negative 	:= FALSE;
			IF Conv_Speed <> M_Velocity THEN
				M_Velocity 	:= Conv_Speed;
				M_Update 	:= TRUE;
			ELSE
				M_Update 	:= FALSE;
			END_IF

			IF Stop_Command OR Error_Command THEN
				State := 3;
			END_IF

			IF Manual_Mode_Trigger THEN
				Man_Mode_OFF 	:= FALSE;
				State 			:= 2;
			END_IF

		2://Manual Motion
			Power_Axis 		:= TRUE;
			M_MoveVelocity	:= FALSE;
			M_Stop 			:= FALSE;
			IF Conv_Left_Man_HMI_Trigger THEN
				M_Jog_Positive := FALSE;
				M_Jog_Negative := TRUE;
			ELSIF Conv_Right_Man_HMI_Trigger THEN
				M_Jog_Positive := TRUE;
				M_Jog_Negative := FALSE;
			ELSE
				M_Jog_Positive := FALSE;
				M_Jog_Negative := FALSE;
			END_IF

			IF NOT Manual_Mode_Trigger THEN
				Power_Axis 		:= FALSE;
				Start_Command 	:= FALSE;
				M_MoveVelocity	:= FALSE;
				M_Jog_Positive 	:= FALSE;
				M_Jog_Negative 	:= FALSE;
				M_Stop 			:= FALSE;
				State 			:= 0;
			END_IF
			IF Stop_Command OR Error_Command THEN
				State := 3;
			END_IF

		3://Stop
			M_MoveVelocity 	:= FALSE;
			M_Stop			:= TRUE;
			M_Jog_Positive 	:= FALSE;
			M_Jog_Negative 	:= FALSE;
			State 			:= 0;
	END_CASE

	Master_Param.Velocity 	:= M_Velocity;
	Master_Param.Jog		:= M_Jog_Param;

	M_Jog_Param.Acceleration 	:= 5000;
	M_Jog_Param.Deceleration 	:= 5000;
	M_Jog_Param.Velocity		:= Conv_Jog_Velocity;
	M_Jog_Param.LowerLimit		:= -1000;
	M_Jog_Param.UpperLimit		:= +1000;

	//Calling Axis Basic Function
	Master(	MpLink 			:= ADR(gAxisBasic_Master),
			Enable 			:= TRUE,
			ErrorReset		:= Reset_Command,
			Parameters 		:= ADR(Master_Param),
			Update			:= M_Update,
			Axis 			:= ADR(gAxis01),
			Power 			:= Power_Axis,
			Home 			:= Home_Axis,
			MoveVelocity 	:= M_MoveVelocity,
			MoveAbsolute 	:= M_MoveAbsolute,
			MoveAdditive 	:= M_MoveAdditive,
			JogPositive 	:= M_Jog_Positive,
			JogNegative		:= M_Jog_Negative,
			Stop 			:= M_Stop);

	M_Active 			:= Master.Active;
	M_Error				:= Master.Error;
	M_Actual_Position	:= Master.Position;
	M_Actual_Velocity 	:= Master.Velocity;
	M_Homed 			:= Master.IsHomed;
	M_Powered 			:= Master.PowerOn;
	M_Stoped 			:= Master.Stopped;

END_PROGRAM

PROGRAM _EXIT
	(* Insert code here *)

END_PROGRAM
```

### Cam.cam
```
CamProfile (NcSwId=ACP10, MasterAxisVelocity=1, MasterAxisAcceleration=0, DefaultCurveType=Polynomial5, MathematicalNotation=true)
  FixPoint (x=0, IsMathX=true, y=0, IsDefinedDy=false, Dy=0, IsMathDy=true, IsDefinedDdy=false, Ddy=0, IsMathDdy=true, IsDefinedDddy=false, Dddy=0, IsMathDddy=true)
  FixPoint (x=0.5, IsMathX=true, y=1, IsDefinedDy=true, Dy=0, IsMathDy=true, IsDefinedDdy=true, Ddy=0, IsMathDdy=true, IsDefinedDddy=false, Dddy=0, IsMathDddy=true)
  FixPoint (x=1, IsMathX=true, y=0, IsDefinedDy=true, Dy=0, IsMathDy=true, IsDefinedDdy=false, Ddy=0, IsMathDdy=true, IsDefinedDddy=false, Dddy=0, IsMathDddy=true)
  Curve (Type=Polynomial5)
    LeftBoundary (IsDefinedDdy=false, Ddy=0, IsMathDdy=true, IsDefinedDddy=false, Dddy=0, IsMathDddy=true)
    RightBoundary (IsDefinedDdy=false, Ddy=0, IsMathDdy=true, IsDefinedDddy=false, Dddy=0, IsMathDddy=true)
    Spline3 (IsContinuous4Derivative=false, IsDefinedSaddlePoint=false, IsDefinedLineAs2ndSegment=false, IsDefinedSlopeOfLine=false, SlopeOfLine=0, IsMathSlopeOfLine=true)
    Supremum (y=1.7e+308, Dy=1.7e+308, IsMathDy=true, Ddy=1.7e+308, IsMathDdy=true, Dddy=1.7e+308, IsMathDddy=true)
    Infimum (y=-1.7e+308, Dy=-1.7e+308, IsMathDy=true, Ddy=-1.7e+308, IsMathDdy=true, Dddy=-1.7e+308, IsMathDddy=true)
  Curve (Type=Polynomial5)
    LeftBoundary (IsDefinedDdy=false, Ddy=0, IsMathDdy=true, IsDefinedDddy=false, Dddy=0, IsMathDddy=true)
    RightBoundary (IsDefinedDdy=false, Ddy=0, IsMathDdy=true, IsDefinedDddy=false, Dddy=0, IsMathDddy=true)
    Spline3 (IsContinuous4Derivative=false, IsDefinedSaddlePoint=false, IsDefinedLineAs2ndSegment=false, IsDefinedSlopeOfLine=false, SlopeOfLine=0, IsMathSlopeOfLine=true)
    Supremum (y=1.7e+308, Dy=1.7e+308, IsMathDy=true, Ddy=1.7e+308, IsMathDdy=true, Dddy=1.7e+308, IsMathDddy=true)
    Infimum (y=-1.7e+308, Dy=-1.7e+308, IsMathDy=true, Ddy=-1.7e+308, IsMathDdy=true, Dddy=-1.7e+308, IsMathDddy=true)
  Cam (LeftBoundaryIndex=0, RightBoundaryIndex=2)
    Supremum (y=1.7e+308, Dy=1.7e+308, IsMathDy=true, Ddy=1.7e+308, IsMathDdy=true, Dddy=1.7e+308, IsMathDddy=true)
    Infimum (y=-1.7e+308, Dy=-1.7e+308, IsMathDy=true, Ddy=-1.7e+308, IsMathDdy=true, Dddy=1.7e+308, IsMathDddy=true)
  ChartExtensions
```

### Cam.cam
```
CamProfile (NcSwId=ACP10, MasterAxisVelocity=1, MasterAxisAcceleration=0, DefaultCurveType=Polynomial5, MathematicalNotation=true)
  FixPoint (x=0, IsMathX=true, y=0, IsDefinedDy=false, Dy=0, IsMathDy=true, IsDefinedDdy=false, Ddy=0, IsMathDdy=true, IsDefinedDddy=false, Dddy=0, IsMathDddy=true)
  FixPoint (x=0.74, IsMathX=true, y=0.1, IsDefinedDy=true, Dy=0.4, IsMathDy=true, IsDefinedDdy=false, Ddy=0, IsMathDdy=true, IsDefinedDddy=false, Dddy=0, IsMathDddy=true)
  FixPoint (x=0.85, IsMathX=true, y=1, IsDefinedDy=true, Dy=0, IsMathDy=true, IsDefinedDdy=true, Ddy=0, IsMathDdy=true, IsDefinedDddy=false, Dddy=0, IsMathDddy=true)
  FixPoint (x=0.95, IsMathX=true, y=0.1, IsDefinedDy=true, Dy=-4.285714286, IsMathDy=true, IsDefinedDdy=false, Ddy=0, IsMathDdy=true, IsDefinedDddy=false, Dddy=0, IsMathDddy=true)
  FixPoint (x=1, IsMathX=true, y=0, IsDefinedDy=false, Dy=0, IsMathDy=true, IsDefinedDdy=false, Ddy=0, IsMathDdy=true, IsDefinedDddy=false, Dddy=0, IsMathDddy=true)
  Curve (Type=Polynomial5)
    LeftBoundary (IsDefinedDdy=false, Ddy=0, IsMathDdy=true, IsDefinedDddy=false, Dddy=0, IsMathDddy=true)
    RightBoundary (IsDefinedDdy=false, Ddy=0, IsMathDdy=true, IsDefinedDddy=false, Dddy=0, IsMathDddy=true)
    Spline3 (IsContinuous4Derivative=false, IsDefinedSaddlePoint=false, IsDefinedLineAs2ndSegment=false, IsDefinedSlopeOfLine=false, SlopeOfLine=0, IsMathSlopeOfLine=true)
    Supremum (y=1.7e+308, Dy=1.7e+308, IsMathDy=true, Ddy=1.7e+308, IsMathDdy=true, Dddy=1.7e+308, IsMathDddy=true)
    Infimum (y=-1.7e+308, Dy=-1.7e+308, IsMathDy=true, Ddy=-1.7e+308, IsMathDdy=true, Dddy=-1.7e+308, IsMathDddy=true)
  Curve (Type=Polynomial5)
    LeftBoundary (IsDefinedDdy=false, Ddy=0, IsMathDdy=true, IsDefinedDddy=false, Dddy=0, IsMathDddy=true)
    RightBoundary (IsDefinedDdy=false, Ddy=0, IsMathDdy=true, IsDefinedDddy=false, Dddy=0, IsMathDddy=true)
    Spline3 (IsContinuous4Derivative=false, IsDefinedSaddlePoint=false, IsDefinedLineAs2ndSegment=false, IsDefinedSlopeOfLine=false, SlopeOfLine=0, IsMathSlopeOfLine=true)
    Supremum (y=1.7e+308, Dy=1.7e+308, IsMathDy=true, Ddy=1.7e+308, IsMathDdy=true, Dddy=1.7e+308, IsMathDddy=true)
    Infimum (y=-1.7e+308, Dy=-1.7e+308, IsMathDy=true, Ddy=-1.7e+308, IsMathDdy=true, Dddy=-1.7e+308, IsMathDddy=true)
  Curve (Type=Polynomial5)
    LeftBoundary (IsDefinedDdy=false, Ddy=0, IsMathDdy=true, IsDefinedDddy=false, Dddy=0, IsMathDddy=true)
    RightBoundary (IsDefinedDdy=false, Ddy=0, IsMathDdy=true, IsDefinedDddy=false, Dddy=0, IsMathDddy=true)
    Spline3 (IsContinuous4Derivative=false, IsDefinedSaddlePoint=false, IsDefinedLineAs2ndSegment=false, IsDefinedSlopeOfLine=false, SlopeOfLine=0, IsMathSlopeOfLine=true)
    Supremum (y=1.7e+308, Dy=1.7e+308, IsMathDy=true, Ddy=1.7e+308, IsMathDdy=true, Dddy=1.7e+308, IsMathDddy=true)
    Infimum (y=-1.7e+308, Dy=-1.7e+308, IsMathDy=true, Ddy=-1.7e+308, IsMathDdy=true, Dddy=-1.7e+308, IsMathDddy=true)
  Curve (Type=Polynomial5)
    LeftBoundary (IsDefinedDdy=false, Ddy=0, IsMathDdy=true, IsDefinedDddy=false, Dddy=0, IsMathDddy=true)
    RightBoundary (IsDefinedDdy=false, Ddy=0, IsMathDdy=true, IsDefinedDddy=false, Dddy=0, IsMathDddy=true)
    Spline3 (IsContinuous4Derivative=false, IsDefinedSaddlePoint=false, IsDefinedLineAs2ndSegment=false, IsDefinedSlopeOfLine=false, SlopeOfLine=0, IsMathSlopeOfLine=true)
    Supremum (y=1.7e+308, Dy=1.7e+308, IsMathDy=true, Ddy=1.7e+308, IsMathDdy=true, Dddy=1.7e+308, IsMathDddy=true)
    Infimum (y=-1.7e+308, Dy=-1.7e+308, IsMathDy=true, Ddy=-1.7e+308, IsMathDdy=true, Dddy=-1.7e+308, IsMathDddy=true)
  Cam (LeftBoundaryIndex=0, RightBoundaryIndex=4)
    Supremum (y=1.7e+308, Dy=1.7e+308, IsMathDy=true, Ddy=1.7e+308, IsMathDdy=true, Dddy=1.7e+308, IsMathDddy=true)
    Infimum (y=-1.7e+308, Dy=-1.7e+308, IsMathDy=true, Ddy=-1.7e+308, IsMathDdy=true, Dddy=1.7e+308, IsMathDddy=true)
  ChartExtensions
```

### Program Logical/Output_Bridge

#### Main.st
```iecst
PROGRAM _INIT
	(* Insert code here *)

END_PROGRAM

PROGRAM _CYCLIC
	(* Insert code here *)
	IF NOT Start_Command THEN
		M_Actual_Velocity := 0;
		S_Actual_Velocity := 0;
	END_IF

	IF DiagCpuIsSimulated() THEN
		ComTCP_SimOutputs.Green_light_Key 	:= DI3.LED_Light;
		ComTCP_SimOutputs.Stop_light_Key 	:= DI4.LED_Light;
		ComTCP_SimOutputs.Yellow_light_Key 	:= DI5.LED_Light;
		ComTCP_SimOutputs.White_light_Key	:= DI6.LED_Light; //it will display red on real setup
		LED_DI1_HMI 						:= DI1.LED_Light;
		LED_DI2_HMI 						:= DI2.LED_Light;
		LED_DI3_HMI 						:= DI3.LED_Light;
		LED_DI4_HMI 						:= DI4.LED_Light;
		LED_DI5_HMI 						:= DI5.LED_Light;
		LED_DI6_HMI 						:= DI6.LED_Light;
		Dis_Conv_Speed_HMI 					:= LREAL_TO_REAL(M_Actual_Velocity)/10;
		Dis_Cut_Speed_HMI 					:= LREAL_TO_REAL(S_Actual_Velocity)/10;

		//Master
		ComTCP_SimOutputs.Shaft_0_ACT_POS 	:= LREAL_TO_REAL(M_Actual_Position);

		//Slave
		ComTCP_SimOutputs.Shaft_1_ACT_POS 	:= LREAL_TO_REAL(S_Actual_Position);

	ELSE
		LED_DI1_HMI 		:= DI1.LED_Light;
		LED_DI2_HMI	 		:= DI2.LED_Light;
		LED_DI3_HMI 		:= DI3.LED_Light;
		LED_DI4_HMI 		:= DI4.LED_Light;
		LED_DI5_HMI 		:= DI5.LED_Light;
		LED_DI6_HMI 		:= DI6.LED_Light;
		Dis_Conv_Speed_HMI 	:= LREAL_TO_REAL(M_Actual_Velocity)/10;
		Dis_Cut_Speed_HMI 	:= LREAL_TO_REAL(S_Actual_Velocity)/10;

		//Hardware
		Display 			:= REAL_TO_INT((LREAL_TO_REAL(M_Actual_Velocity)/10));

	END_IF

END_PROGRAM

PROGRAM _EXIT
	(* Insert code here *)

END_PROGRAM
```

### Program Logical/PLCopen

#### Variables.var
```iecst
VAR
	MC_Power_0 : MC_Power;
	MC_Home_0 : MC_Home;
	MC_Stop_0 : MC_Stop;
	MC_ReadStatus_0 : MC_ReadStatus;
	MC_MoveVelocity_0 : MC_MoveVelocity;
	MC_MoveAdditive_0 : MC_MoveAdditive;
	MC_MoveAbsolute_0 : MC_MoveAbsolute;
	MC_ReadActualPosition_0 : MC_ReadActualPosition;
	MC_ReadActualVelocity_0 : MC_ReadActualVelocity;
	MC_Reset_0 : MC_Reset;
	MyGenericAxisBasicFB_Master : MyGenericAxisBasicFB;
END_VAR
```

#### Main.st
```iecst
PROGRAM _INIT
	(* Insert code here *)

END_PROGRAM

PROGRAM _CYCLIC

	MyGenericAxisBasicFB_Master();

	MC_Power_0.Axis := ADR(gAxis01);
	MC_Power_0();

	MC_Home_0 			(Axis := ADR(gAxis01));
	MC_Stop_0			(Axis := ADR(gAxis01));
	MC_ReadStatus_0		(Axis := ADR(gAxis01));
	MC_MoveVelocity_0	(Axis := ADR(gAxis01));
	MC_MoveAdditive_0	(Axis := ADR(gAxis01));
	MC_MoveAbsolute_0	(Axis := ADR(gAxis01));
	MC_ReadActualPosition_0(Axis := ADR(gAxis01));
	MC_ReadActualVelocity_0(Axis := ADR(gAxis01));
	MC_Reset_0			(Axis := ADR(gAxis01));

END_PROGRAM

PROGRAM _EXIT
	(* Insert code here *)

END_PROGRAM
```

### Program Logical/Slave

#### Variables.var
```iecst
VAR
	State : USINT := 0;
	Slave_Param : MpAxisBasicParType;
	Coupling_Param : MpAxisCouplingParType;
	S_MoveVelocity : BOOL;
	S_MoveAbsolute : BOOL;
	S_MoveAdditive : BOOL;
	C_Synced : BOOL;
	S_Stop : BOOL;
	S_Jog_Param : MpAxisJogType;
	S_Jog_Positive : BOOL;
	S_Jog_Negative : BOOL;
	S_Position : REAL;
	S_Velocity : REAL;
	S_Direction : MpAxisMoveDirectionEnum;
END_VAR
```

#### Main.st
```iecst
PROGRAM _INIT
	(* Insert code here *)
	Coupling_Param.RatioDenominator := 360.0;
	Coupling_Param.RatioNumerator 	:= 360.0;

	//Cam graph to be linked
	Coupling_Param.Cam.CamTable[0] 	:= 'MyCam';
	Coupling_Param.Cam.CamTable[1]	:= 'MyCamBis';

	Coupling_Param.Cam.CamTableID 	:= 1;

END_PROGRAM

PROGRAM _CYCLIC

	CASE State OF
		0: // Synced Cutting using CAM
			IF C_Synced THEN
				Done_Cut := TRUE;
			END_IF

			IF Manual_Mode_Trigger THEN
				Man_Mode_OFF 	:= FALSE;
				State 			:= 1;
			END_IF

		1: //Manual Mode
			Power_Axis 		:= TRUE;
			S_MoveVelocity 	:= FALSE;
			S_Stop 			:= FALSE;
			IF Blade_Down_Man_HMI_Trigger THEN
				S_Jog_Positive := FALSE;
				S_Jog_Negative := TRUE;
			ELSIF Blade_Up_Man_HMI_Trigger THEN
				S_Jog_Positive := TRUE;
				S_Jog_Negative := FALSE;
			ELSE
				S_Jog_Positive := FALSE;
				S_Jog_Negative := FALSE;
			END_IF
			IF NOT Manual_Mode_Trigger THEN
				IF S_Actual_Position <> 0.0 THEN
					S_Velocity 		:= 50;
					S_MoveAbsolute 	:= TRUE;
					S_Position 		:= 0.0;
					S_Direction 	:= mpAXIS_DIR_SHORTEST_WAY;
					S_MoveVelocity 	:= FALSE;
					S_Jog_Positive 	:= FALSE;
					S_Jog_Negative 	:= FALSE;
					S_Stop 			:= FALSE;
				END_IF
				IF S_Actual_Position = 0.0 THEN
					Man_Mode_OFF 	:= TRUE;
					Power_Axis 		:= FALSE;
					S_MoveVelocity 	:= FALSE;
					S_MoveAbsolute 	:= FALSE;
					S_Jog_Positive 	:= FALSE;
					S_Jog_Negative 	:= FALSE;
					S_Stop 			:= FALSE;
					State 			:= 0;
				END_IF
			END_IF

	END_CASE

	Slave_Param.Jog 			:= S_Jog_Param;
	Slave_Param.Acceleration 	:= 1000;
	Slave_Param.Deceleration 	:= 1000;
	Slave_Param.Velocity 		:= S_Velocity;
	Slave_Param.Position 		:= S_Position;
	Slave_Param.Direction 		:= S_Direction;

	S_Jog_Param.Acceleration 	:= 5000;
	S_Jog_Param.Deceleration 	:= 5000;
	S_Jog_Param.Velocity		:= Blade_Jog_Velocity;
	S_Jog_Param.LowerLimit		:= -1000;
	S_Jog_Param.UpperLimit		:= +1000;

	//Calling FSM_AXIS Function
	Slave(	MpLink 			:= ADR(gAxisBasic_Slave),
			Enable 			:= TRUE,
			ErrorReset		:= Reset_Command,
			Parameters 		:= ADR(Slave_Param),
			Axis 			:= ADR(gAxis02),
			Power 			:= Power_Axis,
			Home 			:= Home_Axis,
			MoveVelocity 	:= S_MoveVelocity,
			MoveAbsolute 	:= S_MoveAbsolute,
			MoveAdditive 	:= S_MoveAdditive,
			JogPositive 	:= S_Jog_Positive,
			JogNegative 	:= S_Jog_Negative,
			Stop 			:= S_Stop);

	S_Active 			:= Slave.Active;
	S_Error				:= Slave.Error;
	S_Homed 			:= Slave.IsHomed;
	S_Powered 			:= Slave.PowerOn;
	S_Stoped 			:= Slave.Stopped;

	Coupling(	MpLink 			:= ADR(gAxisBasic_Slave),
				Enable 			:= TRUE,
				Cam 			:= Do_Cut,
				ErrorReset 		:= Reset_Command,
				Gear 			:= 1,
				Parameters 		:= ADR(Coupling_Param),
				MpLinkMaster 	:= ADR(gAxisBasic_Master));

	C_Synced 			:= Coupling.InSync;
	C_Error 			:= Coupling.Error;
	S_Actual_Position 	:= Coupling.Info.SlavePosition;
	S_Actual_Velocity 	:= Coupling.Info.SlaveVelocity;

END_PROGRAM

PROGRAM _EXIT
	(* Insert code here *)

END_PROGRAM
```

Listed in the project but not available here: Logical/Libraries/My_Library/Types.typ, Logical/Libraries/My_Library/Constants.var, Logical/Libraries/My_Library/FSM_LED.st, Logical/Libraries/My_Library/FSM_AXIS.st
